Fanuc KAREL source: kt00406.KL

-- PROVISIONAL review KL for V940-1; original PC SHA256 6ca55cabb3e88c93ea3c71ab5e6560d0f9d8740acb6ffeed1ac539b999248e53
-- Incomplete behavior may be omitted. Consult companion uncertainty JSON. Do not deploy.
PROGRAM KT00406
%NOLOCKGROUP
VAR
  R1 : REAL
  R2 : REAL
  OUT : BOOLEAN
BEGIN
  -- V9_ZERO_TABLE_METADATA_HINT layout=0001; no indexed target words; source/name/runtime held
  -- UNRESOLVED_PC offsets 5-16; opcodes 2E,23
  -- UNRESOLVED_PC offsets 21-32; opcodes 2E,23
  -- UNRESOLVED_PC offsets 37-48; opcodes 2E,23
  -- UNRESOLVED_PC offsets 53-64; opcodes 2E,23
  -- UNRESOLVED_PC offsets 69-88; opcodes 21,21,71,23
  -- UNRESOLVED_PC offsets 93-97; opcodes 7F
END KT00406
